FUNCTION_BLOCK ALR_SPLIT_5 (* SPLIT 1 ALR into 5 ALR (generic FB) Adapter-Ausgang wird nur bei Wertänderung aktualisiert (Event nur bei tatsächlicher Änderung). *)
  (* Standard: 61499-2; Description: Copyright (c) 2025 HR Agrartechnik GmbH This program and the accompanying materials are made available under the terms of the Eclipse Public License 2.0 which is available at https://www.eclipse.org/legal/epl-2.0/ SPDX-License-Identifier: EPL-2.0 *)
  (* Version 1.0, 2025-01-24, Franz Höpfinger, HR Agrartechnik GmbH *)
  PACKAGE adapter::events::unidirectional;
  IMPORT eclipse4diac::core::GenericClassName;
  {SET_ATTRIBUTE(eclipse4diac::core::GenericClassName, 'GEN_ALR_SPLIT')}
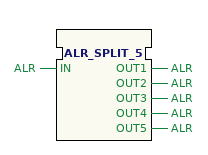
  SOCKETS
    IN : adapter::types::unidirectional::ALR;
  END_SOCKETS
  PLUGS
    OUT1 : adapter::types::unidirectional::ALR;
    OUT2 : adapter::types::unidirectional::ALR;
    OUT3 : adapter::types::unidirectional::ALR;
    OUT4 : adapter::types::unidirectional::ALR;
    OUT5 : adapter::types::unidirectional::ALR;
  END_PLUGS
END_FUNCTION_BLOCK
